% RSLogix 500 project TOOL OPERATION_BAK036.RSS, saved by version 8.10.00.18 %
PROJECT "UNTITLED"    % processor: MicroLogix 1200 %

PROGRAM FILES
  LAD 2   9 rungs

DATA FILES
  O0 OUTPUT  4 elements
  I1 INPUT  4 elements
  S2 STATUS  66 elements
  B3 BINARY  1 elements
  T4 TIMER  1 elements
  C5 COUNTER  1 elements
  R6 CONTROL  1 elements
  N7 INTEGER  1 elements

LADDER 2
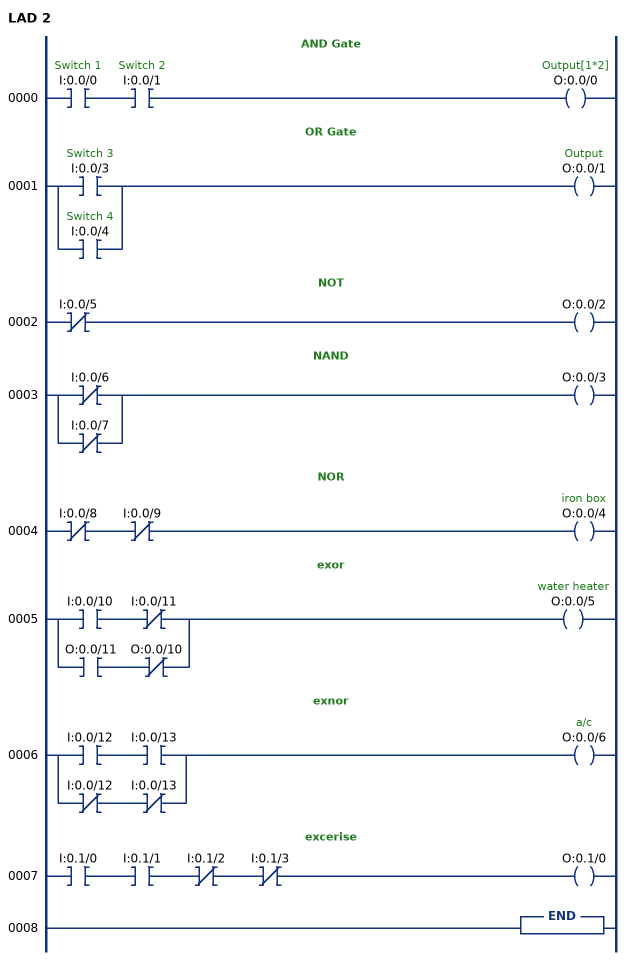
% Rung: 0 %
% TITLE: AND Gate %
SOR XIC I:0.0/0 XIC I:0.0/1 OTE O:0.0/0 EOR
%   I:0.0/0  "Switch 1" %
%   I:0.0/1  "Switch 2" %
%   O:0.0/0  "Output[1*2]" %
% Rung: 1 %
% TITLE: OR Gate %
SOR BST XIC I:0.0/3 NXB XIC I:0.0/4 BND OTE O:0.0/1 EOR
%   I:0.0/3  "Switch 3" %
%   I:0.0/4  "Switch 4" %
%   O:0.0/1  "Output" %
% Rung: 2 %
% TITLE: NOT %
SOR XIO I:0.0/5 OTE O:0.0/2 EOR
% Rung: 3 %
% TITLE: NAND %
SOR BST XIO I:0.0/6 NXB XIO I:0.0/7 BND OTE O:0.0/3 EOR
% Rung: 4 %
% TITLE: NOR %
SOR XIO I:0.0/8 XIO I:0.0/9 OTE O:0.0/4 EOR
%   O:0.0/4  "iron box" %
% Rung: 5 %
% TITLE: exor %
SOR BST XIC I:0.0/10 XIO I:0.0/11 NXB XIC O:0.0/11 XIO O:0.0/10 BND OTE O:0.0/5 EOR
%   O:0.0/5  "water heater" %
% Rung: 6 %
% TITLE: exnor %
SOR BST XIC I:0.0/12 XIC I:0.0/13 NXB XIO I:0.0/12 XIO I:0.0/13 BND OTE O:0.0/6 EOR
%   O:0.0/6  "a/c" %
% Rung: 7 %
% TITLE: excerise %
SOR XIC I:0.1/0 XIC I:0.1/1 XIO I:0.1/2 XIO I:0.1/3 OTE O:0.1/0 EOR
% Rung: 8 %
SOR END EOR

OTHER DOCUMENTED ADDRESSES
  I:0.0/2  "Switch 3"
